// TwinCAT 3 PLC project
// Title: Demo
// Company: Robsen Robotics
// ProjectVersion: 1.0.0.0
// libraries:
//   Tc2_Standard, * (Beckhoff Automation GmbH)
//   Tc2_System, * (Beckhoff Automation GmbH)
//   Tc3_Module, * (Beckhoff Automation GmbH)
// project tree:
//   POUs/ FB_Conveyor.TcPOU, MAIN.TcPOU, F_IsError.TcPOU
//   DUTs/ E_ConveyorState.TcDUT, ST_ConveyorConfig.TcDUT
//   GVLs/ GVL_Main.TcGVL
//   ITfs/ I_Device.TcIO
// real-time tasks:
//   TASK PlcTask: cycle T#10ms, priority 20, ADS port 350

// ---- DUTs/E_ConveyorState.TcDUT
TYPE E_ConveyorState :
(
    Idle := 0,
    Starting,
    Running,
    Fault
);
END_TYPE

// ---- DUTs/ST_ConveyorConfig.TcDUT
TYPE ST_ConveyorConfig :
STRUCT
    tStartupDelay : TIME := T#200MS;
    rMaxSpeed : REAL := 100.0;
    sName : STRING(63);
END_STRUCT
END_TYPE

// ---- GVLs/GVL_Main.TcGVL
{attribute 'qualified_only'}
VAR_GLOBAL
    rMaxSpeed : REAL := 250.0;
    bEmergencyStop : BOOL;
END_VAR
VAR_GLOBAL CONSTANT
    nMAX_AXES : UDINT := 8;
END_VAR

// ---- ITfs/I_Device.TcIO
INTERFACE I_Device

METHOD Init : BOOL
VAR_INPUT
    nId : UDINT;
END_VAR
END_METHOD

METHOD Reset
END_METHOD

END_INTERFACE

// ---- POUs/FB_Conveyor.TcPOU
FUNCTION_BLOCK FB_Conveyor EXTENDS FB_Base IMPLEMENTS I_Device
VAR_INPUT
    bEnable : BOOL;
    rSetSpeed : REAL := 0.0;
END_VAR
VAR_OUTPUT
    bRunning : BOOL;
END_VAR
VAR
    fbMotor : FB_Motor;
    tonDelay : TON;
    eState : E_ConveyorState;
    stConfig : ST_ConveyorConfig;
    _rSpeed : REAL;
END_VAR

tonDelay(IN := bEnable, PT := stConfig.tStartupDelay);
fbMotor(bEnable := bEnable);
bRunning := fbMotor.bActive AND NOT F_IsError(fbMotor);
UpdateState();

METHOD Start : BOOL
VAR_INPUT
    rSpeed : REAL;
END_VAR
IF rSpeed > GVL_Main.rMaxSpeed THEN
    rSpeed := GVL_Main.rMaxSpeed;
END_IF
fbMotor.SetSpeed(rSpeed := rSpeed);
Start := TRUE;
END_METHOD

METHOD PRIVATE UpdateState
CASE eState OF
    E_ConveyorState.Idle:
        IF bEnable THEN
            eState := E_ConveyorState.Starting;
        END_IF
    E_ConveyorState.Starting:
        tonDelay(IN := TRUE, PT := T#500MS);
        IF tonDelay.Q THEN
            eState := E_ConveyorState.Running;
        END_IF
END_CASE
END_METHOD

ACTION A_Reset:
eState := E_ConveyorState.Idle;
bRunning := FALSE;
END_ACTION

PROPERTY Speed : REAL
GET
Speed := _rSpeed;
END_GET
SET
_rSpeed := Speed;
END_SET
END_PROPERTY

END_FUNCTION_BLOCK

// ---- POUs/F_IsError.TcPOU
FUNCTION F_IsError : BOOL
VAR_INPUT
    fb : FB_Motor;
END_VAR

F_IsError := fb.nErrorId <> 0;

END_FUNCTION

// ---- POUs/MAIN.TcPOU
PROGRAM MAIN
VAR
    fbConveyor : FB_Conveyor;
    bStartCmd : BOOL;
    nCycles : UDINT;
END_VAR

fbConveyor(bEnable := bStartCmd AND NOT GVL_Main.bEmergencyStop);
IF fbConveyor.Start(rSpeed := 50.0) THEN
    nCycles := nCycles + 1;
END_IF

END_PROGRAM
